FUNCTION GetBit : BOOL
VAR_INPUT
	data			: ANY;
	bitIndex		: UDINT;
END_VAR
VAR
	byteIndex		: UDINT;
	bitNumber		: UDINT;
END_VAR

byteIndex := bitIndex / 8;
bitNumber := bitIndex MOD 8;
GetBit := BYTE_TO_BOOL(SHR(data.pValue[byteIndex], bitNumber) AND 16#01);

END_FUNCTION

(* stored: Version 1.1.0.1
   POU GetBit: Id {42277088-d5a2-0a8f-1797-6626b69cb432}, SpecialFunc None *)
